// TIA Portal V18 export
FUNCTION "Block_1" : Void   // FC1, LAD
{ S7_Optimized_Access := 'TRUE' }
VERSION : 0.1
// stored: AutoNumber true, IsIECCheckEnabled false, SetENOAutomatically false, UDAEnableTagReadback false
BEGIN

REGION Network 1: Network1-addin sss
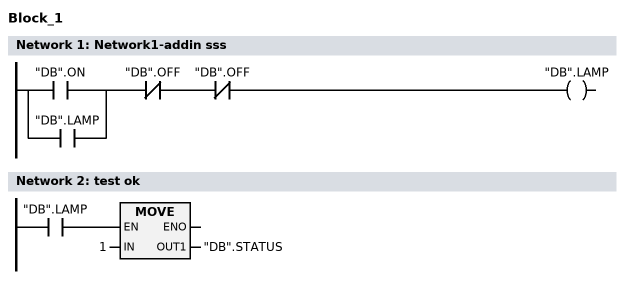
   RUNG wire#powerrail
      Contact( "DB".ON )
      wire#w1
      I_Contact( "DB".OFF )
      I_Contact( "DB".OFF )
      Coil( "DB".LAMP )
   END_RUNG
   RUNG wire#powerrail
      Contact( "DB".LAMP )
   END_RUNG wire#w1
   // the same network as SCL:
   "DB".LAMP := ("DB".ON OR "DB".LAMP) AND NOT "DB".OFF AND NOT "DB".OFF;
END_REGION

REGION Network 2: test ok
   RUNG wire#powerrail
      Contact( "DB".LAMP )
      Move(in := 1, out1 => "DB".STATUS)
   END_RUNG
   // the same network as SCL:
   IF "DB".LAMP THEN "DB".STATUS := 1; END_IF;
END_REGION

REGION Network 3: test
END_REGION
END_FUNCTION
